// SIMATIC S7-200 project (STEP 7-Micro/WIN), CPU 221 REL 01.10

SYMBOL_TABLE USR1
Always_On        SM0.0    // This bit is always on.
On_Pushbutton    I0.0     // Pushbutton turns the light on.
Light            Q0.0     // Light is lit when output is set.
Timer_30s        T37      // Timer turns the light off after 30 seconds.
END_SYMBOL_TABLE

ORGANIZATION_BLOCK MAIN:OB1
TITLE=
//  阶梯灯的定时点亮
//  ***概述***
// 本程序用来点亮阶梯灯。不同层上的ON按钮都被接到控制输入端I0.0。当按下
// I0.0的ON按钮，则输出端Q0.0的灯发光30秒，如果在这段时间内又一次按ON按钮，
// 则时间间隔又得从头开始。这样可确保在最后一次按ON按钮，在30秒内灯光不会熄灭。
// ***程序和注释***
// 如果按ON按钮，使输入的I0.0的ON信号有效（I0.0=1），则定时器位T37复位（T37=0)。
// 因而定时器T37从头开始计时。与此同时，输出Q0.0被置位（Q0.0=1，灯亮）。当计足30
// 秒，定时器位T37置位（T37=1),那将又一次使输出Q0.0为OFF（Q0.0=0,灯灭）。
// 题目：定时
// 
BEGIN
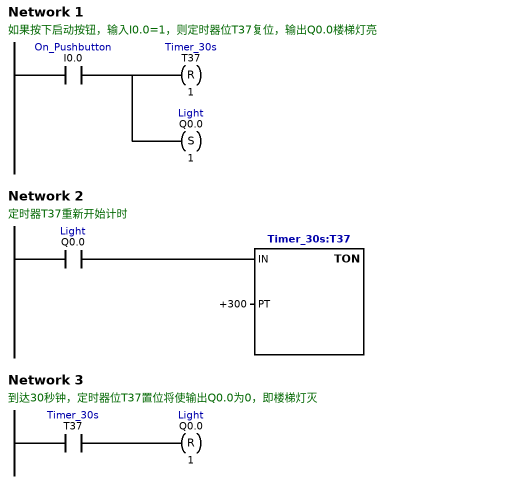
Network 1
// 如果按下启动按钮，输入I0.0=1，则定时器位T37复位，输出Q0.0楼梯灯亮
// 若一个按钮被按下(I0.0=1),则
// 定时器T37复位(T37=0)
// 开灯(Q0.0=1)
// (network saved uncompiled; LAD cells follow)
// row 0: c0 -| |- On_Pushbutton:I0.0 v  c1 -(R) Timer_30s:T37, 1
// row 1: c0 ^  c1 -(S) Light:Q0.0, 1
Network 2
// 定时器T37重新开始计时
//特殊存储标记位SM0.0总是1
//让定时器计时30秒(100ms*300=30s)
LD     Light:Q0.0
TON    Timer_30s:T37, +300
Network 3
// 到达30秒钟，定时器位T37置位将使输出Q0.0为0，即楼梯灯灭
//若30秒时间到，则
// 关灯(Q0.0=0)
LD     Timer_30s:T37
R      Light:Q0.0, 1
Network 4 //  主程序结束
// MEND				
// 
END_ORGANIZATION_BLOCK
